Staubli VAL3: iFluor.pgx

public program iFluor(num& nNum[] (dimensions=1))
begin
  if (dioGet(iFluorClosed)==0) and (dioGet(iFluorOpen)==1)
    nNum=1
  endIf
  if (dioGet(iFluorClosed)==1) and (dioGet(iFluorOpen)==0)
    nNum=0
  endIf
end
